Yaskawa INFORM job: OBR_-90_180.JBI

/JOB
//NAME OBR_-90_180
//POS
///NPOS 0,0,1,0,0,0
///TOOL 0
///POSTYPE PULSE
///PULSE
EC00000=-798156,1112951
//INST
///DATE 2024/03/05 20:16
///ATTR SC,RW
///GROUP1 ST1
NOP
MOVJ EC00000 VJ=100.00
END
